PROGRAM PrgMqttCom
VAR
	fbMqttClient : FB_IotMqttClient;
	bSetParameter : BOOL := TRUE;
	bConnect : BOOL := TRUE;
	
	(* published message *)
	sTopicPub : STRING(255) := 'Test/Text_To_Speech';
	sPayloadPub : STRING(255);
	
	hrErrorOccurred : HRESULT; // contains the latest occurred error
END_VAR

IF bSetParameter THEN
	bSetParameter := FALSE;
	fbMqttClient.sHostName:= '192.168.1.205';
	fbMqttClient.nHostPort:= 1883;
	fbMqttClient.sTopicPrefix:= ''; 
END_IF

sPayloadPub := GVL.message_pub;

IF NOT(GVL.flag_pub) THEN
	fbMqttClient.Execute(bConnect);
	IF fbMqttClient.bError THEN
		hrErrorOccurred := fbMqttClient.hrErrorCode;
	END_IF
	IF fbMqttClient.bConnected THEN
		GVL.flag_pub := TRUE;
	END_IF
END_IF

IF GVL.flag_pub THEN
		fbMqttClient.Publish(	sTopic:= sTopicPub, 
								pPayload:= ADR(sPayloadPub), nPayloadSize:= LEN2(ADR(sPayloadPub)), 
								eQoS:= TcIotMqttQos.AtMostOnceDelivery, bRetain:= FALSE, bQueue:= FALSE );
		IF fbMqttClient.bError THEN
			hrErrorOccurred := fbMqttClient.hrErrorCode;
		END_IF
END_IF

END_PROGRAM

(* stored: Version 1.1.0.1, ProductVersion 3.1.4024.2
   POU PrgMqttCom: Id {3b2be917-83cc-458a-ab8b-8055a76a6ef3}, SpecialFunc None *)
